Universal Robots PolyScope program: swing2.urp

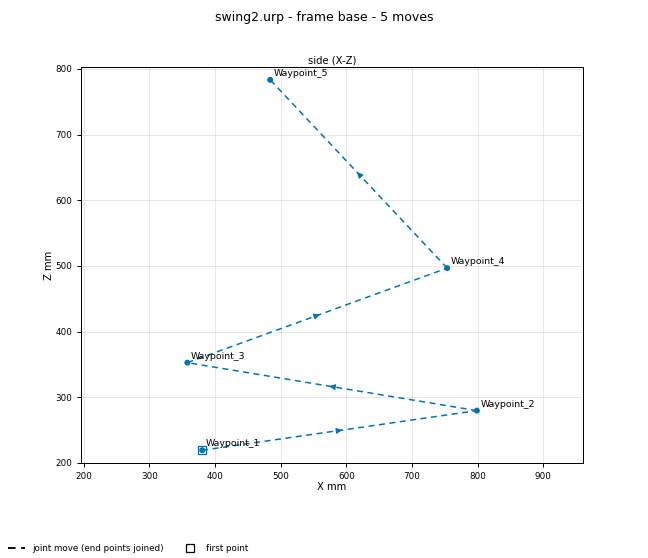
[picture p0: tool path of swing2.urp in frame base, 5 of 5 moves have a stored position in this frame; points joined in program order, loops and branches not executed]
Program swing2 (installation=default directory=/programs createdIn=5.2.0.61336 lastSavedIn=5.2.0.61336 robotSerialNumber=20195500451)
Calibrated DH parameters: a=[0.00002, -0.231658, -0.317125, 0.000011, 0.000055, 0]; d=[0.162082, 123.190176, -180.284242, 57.22734, 0.099524, 0.09934]; alpha=[1.569304, 0.00289, 0.004025, 1.569925, -1.569026, 0]; deltaTheta=[0, 0.993923, 4.662183, 0.627072, 0.000001, 0]
Robot Program (runOnlyOnce=true)
  MoveJ speed 100 deg/s, acceleration 100 deg/s^2 (useActiveTCP=true) feature=Base
    Waypoint Waypoint_1: motionParameters(nextMotionTime=2); TCP in base x=380.392 y=-132.813 z=219.178 mm, rx=1.3369 ry=1.3411 rz=1.1208 rad; joints [-0.005, -90, -130.072, -150.002, -89.999, 0] deg; TCP offset x=0 y=0 z=0 mm, rx=0 ry=0 rz=0 rad
    Waypoint Waypoint_2: motionParameters(nextMotionTime=0.5); TCP in base x=798.729 y=-134.28 z=279.511 mm, rx=1.0269 ry=1.0326 rz=1.3109 rad; joints [0, -135.326, -60.789, -150, -90, 0] deg; TCP offset x=0 y=0 z=0 mm, rx=0 ry=0 rz=0 rad
    Wait Sleep waitTime=0.3
    Waypoint Waypoint_3: motionParameters(nextMotionTime=0.5); TCP in base x=357.678 y=-132.654 z=352.61 mm, rx=1.0793 ry=1.0843 rz=1.2862 rad; joints [0, -72.793, -127.261, -150, -90, 0] deg; TCP offset x=0 y=0 z=0 mm, rx=0 ry=0 rz=0 rad
    Wait Sleep waitTime=0.2
    Waypoint Waypoint_4: motionParameters(nextMotionTime=0.5); TCP in base x=753.519 y=-134.009 z=496.621 mm, rx=0.7982 ry=0.8037 rz=1.4152 rad; joints [0, -122.047, -56.79, -150, -90, 0] deg; TCP offset x=0 y=0 z=0 mm, rx=0 ry=0 rz=0 rad
    Waypoint Waypoint_5: motionParameters(nextMotionTime=0.4 blendRadius=0.05); TCP in base x=483.883 y=-133.125 z=783.376 mm, rx=0.0066 ry=0.011 rz=1.5698 rad; joints [0.004, -90.54, -75.001, -105, -89.999, 0] deg
